// TIA Portal V19 export
VAR_GLOBAL   // PLC tag table "A03_301"
   A0301_Rulliera_Phc_1 AT %I201.2 : Bool;   // 1445BF1
   A0301_Rulliera_Phc_2 AT %I201.3 : Bool;   // 1445SQ1/SQ2/SQ3/SQ4
   A0301_Rulliera_Phc_3 AT %I201.4 : Bool;   // 1445SQ5/SQ6/SQ7/SQ8
   A0301_Rulliera_Phc_4 AT %I201.5 : Bool;   // 1446SQ1/SQ2/SQ3/SQ4
   A0301_Rulliera_Phc_5 AT %I201.6 : Bool;   // 1446BF1
   A0301_Spintore_1_Verticale_Ls_Rest AT %I201.7 : Bool;   // 1450SQ1
   A0301_Spintore_1_Verticale_V_Rest AT %Q210.0 : Bool;   // 1450YV1
   A0301_Spintore_1_Verticale_V_Work AT %Q210.1 : Bool;   // 1450YV2
   A0301_Spintore_1_Laterale_Ls_Rest AT %I202.0 : Bool;   // 1450SQ2
   A0301_Spintore_1_Laterale_V_Rest AT %Q210.2 : Bool;   // 1450YV3
   A0301_Spintore_1_Laterale_V_Work AT %Q210.3 : Bool;   // 1450YV4
   A0301_Spintore_1_Laterale_Ls_Work AT %I202.1 : Bool;   // 1450SQ3
   A0301_Spintore_2_Verticale_Ls_Rest AT %I202.2 : Bool;   // 1451SQ1
   A0301_Spintore_2_Verticale_V_Rest AT %Q210.4 : Bool;   // 1451YV1
   A0301_Spintore_2_Verticale_V_Work AT %Q210.5 : Bool;   // 1451YV2
   A0301_Spintore_2_Laterale_Ls_Rest AT %I202.3 : Bool;   // 1451SQ2
   A0301_Spintore_2_Laterale_V_Rest AT %Q210.6 : Bool;   // 1451YV3
   A0301_Spintore_2_Laterale_V_Work AT %Q210.7 : Bool;   // 1451YV4
   A0301_Spintore_2_Laterale_Ls_Work AT %I202.4 : Bool;   // 1451SQ3
   A0301_Spintore_3_Verticale_Ls_Rest AT %I202.5 : Bool;   // 1452SQ1
   A0301_Spintore_3_Verticale_V_Rest AT %Q211.0 : Bool;   // 1452YV1
   A0301_Spintore_3_Verticale_V_Work AT %Q211.1 : Bool;   // 1452YV2
   A0301_Spintore_3_Laterale_Ls_Rest AT %I202.6 : Bool;   // 1452SQ2
   A0301_Spintore_3_Laterale_V_Rest AT %Q211.2 : Bool;   // 1452YV3
   A0301_Spintore_3_Laterale_V_Work AT %Q211.3 : Bool;   // 1452YV4
   A0301_Spintore_3_Laterale_Ls_Work AT %I202.7 : Bool;   // 1452SQ3
   A0301_Spintore_4_Verticale_Ls_Rest AT %I203.0 : Bool;   // 1453SQ1
   A0301_Spintore_4_Verticale_V_Rest AT %Q211.4 : Bool;   // 1453YV1
   A0301_Spintore_4_Verticale_V_Work AT %Q211.5 : Bool;   // 1453YV2
   A0301_Spintore_4_Laterale_Ls_Rest AT %I203.1 : Bool;   // 1453SQ2
   A0301_Spintore_4_Laterale_V_Rest AT %Q211.6 : Bool;   // 1453YV3
   A0301_Spintore_4_Laterale_V_Work AT %Q211.7 : Bool;   // 1453YV4
   A0301_Spintore_4_Laterale_Ls_Work AT %I203.2 : Bool;   // 1453SQ3
   A0301_Spintore_5_Verticale_Ls_Rest AT %I203.3 : Bool;   // 1454SQ1
   A0301_Spintore_5_Verticale_V_Rest AT %Q212.0 : Bool;   // 1454YV1
   A0301_Spintore_5_Verticale_V_Work AT %Q212.1 : Bool;   // 1454YV2
   A0301_Spintore_5_Laterale_Ls_Rest AT %I203.4 : Bool;   // 1454SQ2
   A0301_Spintore_5_Laterale_V_Rest AT %Q212.2 : Bool;   // 1454YV3
   A0301_Spintore_5_Laterale_V_Work AT %Q212.3 : Bool;   // 1454YV4
   A0301_Spintore_5_Laterale_Ls_Work AT %I203.5 : Bool;   // 1454SQ3
   A0301_Spintore_6_Verticale_Ls_Rest AT %I203.6 : Bool;   // 1455SQ1
   A0301_Spintore_6_Verticale_V_Rest AT %Q212.4 : Bool;   // 1455YV1
   A0301_Spintore_6_Verticale_V_Work AT %Q212.5 : Bool;   // 1455YV2
   A0301_Spintore_6_Laterale_Ls_Rest AT %I203.7 : Bool;   // 1455SQ2
   A0301_Spintore_6_Laterale_V_Rest AT %Q212.6 : Bool;   // 1455YV3
   A0301_Spintore_6_Laterale_V_Work AT %Q212.7 : Bool;   // 1455YV4
   A0301_Spintore_6_Laterale_Ls_Work AT %I204.0 : Bool;   // 1455SQ3
   A0301_Scivolo_1_Phc_1 AT %I204.1 : Bool;   // 1470SQ1
   A0301_Scivolo_1_Phc_2 AT %I204.2 : Bool;   // 1470SQ2
   A0301_Scivolo_1_Phc_3 AT %I204.3 : Bool;   // 1470SQ3
   A0301_Scivolo_1_Phc_4 AT %I204.4 : Bool;   // 1470SQ4
   A0301_Cinghia_1_Phc_1 AT %I253.0 : Bool;   // 1510SQ1
   A0301_Cinghia_1_Phc_4 AT %I253.3 : Bool;   // 1510SQ4
   A0301_Cinghia_1_Phc_2 AT %I253.1 : Bool;   // 1510SQ2
   A0301_Cinghia_1_Phc_3 AT %I253.2 : Bool;   // 1510SQ3
   A0301_Cinghia_1_Phc_5 AT %I253.4 : Bool;   // 1510SQ5
   A0301_Cinghia_1_Phc_6 AT %I253.5 : Bool;   // 1510SQ6
   A0301_Cinghia_1_Phc_7 AT %I253.6 : Bool;   // 1510SQ7
   A0301_Cinghia_1_Phc_8 AT %I253.7 : Bool;   // 1510SQ8
   A0301_Cinghia_2_Phc_1 AT %I254.0 : Bool;   // 1511SQ1
   A0301_Cinghia_2_Phc_2 AT %I254.1 : Bool;   // 1511SQ2
   A0301_Cinghia_2_Phc_3 AT %I254.2 : Bool;   // 1511SQ3
   A0301_Cinghia_2_Phc_4 AT %I254.3 : Bool;   // 1511SQ4
   A0301_Cinghia_2_Phc_5 AT %I254.4 : Bool;   // 1511SQ5
   A0301_Cinghia_2_Phc_6 AT %I254.5 : Bool;   // 1511SQ6
   A0301_Cinghia_2_Phc_7 AT %I254.6 : Bool;   // 1511SQ7
   A0301_Cinghia_2_Phc_8 AT %I254.7 : Bool;   // 1511SQ8
   A0301_Cinghia_4_Phc_1 AT %I255.0 : Bool;   // 1513SQ1
   A0301_Cinghia_4_Phc_2 AT %I255.1 : Bool;   // 1513SQ2
   A0301_Cinghia_4_Phc_3 AT %I255.2 : Bool;   // 1513SQ3
   A0301_Cinghia_4_Phc_4 AT %I255.3 : Bool;   // 1513SQ4
   A0301_Cinghia_4_Phc_5 AT %I255.4 : Bool;   // 1513SQ5
   A0301_Cinghia_4_Phc_6 AT %I255.5 : Bool;   // 1513SQ6
   A0301_Cinghia_4_Phc_7 AT %I255.6 : Bool;   // 1513SQ7
   A0301_Cinghia_4_Phc_8 AT %I255.7 : Bool;   // 1513SQ8
   "A0301_CinghiaTrasporto_1.1_Ls_Rest_1" AT %I256.0 : Bool;   // 1530SQ1
   "A0301_CinghiaTrasporto_1.1_Ls_Work_2" AT %I256.1 : Bool;   // 1530SQ2
   "A0301_CinghiaTrasporto_1.1_Ls_Rest_3" AT %I256.2 : Bool;   // 1530SQ3
   "A0301_CinghiaTrasporto_1.1_Ls_Work_4" AT %I256.3 : Bool;   // 1530SQ4
   "A0301_CinghiaTrasporto_1.1_Ls_Rest_5" AT %I256.4 : Bool;   // 1530SQ5
   "A0301_CinghiaTrasporto_1.1_Ls_Work_6" AT %I256.5 : Bool;   // 1530SQ6
   "A0301_CinghiaTrasporto_1.1_Ls_Rest_7" AT %I256.6 : Bool;   // 1530SQ7
   "A0301_CinghiaTrasporto_1.2_Ls_Rest_1" AT %I257.0 : Bool;   // 1531SQ1
   "A0301_CinghiaTrasporto_1.2_Ls_Work_2" AT %I257.1 : Bool;   // 1531SQ2
   "A0301_CinghiaTrasporto_1.2_Ls_Rest_3" AT %I257.2 : Bool;   // 1531SQ3
   "A0301_CinghiaTrasporto_1.2_Ls_Work_4" AT %I257.3 : Bool;   // 1531SQ4
   "A0301_CinghiaTrasporto_1.2_Ls_Rest_5" AT %I257.4 : Bool;   // 1531SQ5
   "A0301_CinghiaTrasporto_2.1_Ls_Rest_1" AT %I258.0 : Bool;   // 1532SQ1
   "A0301_CinghiaTrasporto_2.1_Ls_Work_2" AT %I258.1 : Bool;   // 1532SQ2
   "A0301_CinghiaTrasporto_2.1_Ls_Rest_3" AT %I258.2 : Bool;   // 1532SQ3
   "A0301_CinghiaTrasporto_2.1_Ls_Work_4" AT %I258.3 : Bool;   // 1532SQ4
   "A0301_CinghiaTrasporto_2.1_Ls_Rest_5" AT %I258.4 : Bool;   // 1532SQ5
   "A0301_CinghiaTrasporto_2.1_Ls_Work_6" AT %I258.5 : Bool;   // 1532SQ6
   "A0301_CinghiaTrasporto_2.1_Ls_Rest_7" AT %I258.6 : Bool;   // 1532SQ7
   "A0301_CinghiaTrasporto_2.2_Ls_Rest_1" AT %I259.0 : Bool;   // 1533SQ1
   "A0301_CinghiaTrasporto_2.2_Ls_Work_2" AT %I259.1 : Bool;   // 1533SQ2
   "A0301_CinghiaTrasporto_2.2_Ls_Rest_3" AT %I259.2 : Bool;   // 1533SQ3
   "A0301_CinghiaTrasporto_2.2_Ls_Work_4" AT %I259.3 : Bool;   // 1533SQ4
   "A0301_CinghiaTrasporto_2.2_Ls_Rest_5" AT %I259.4 : Bool;   // 1533SQ5
   "A0301_CinghiaTrasporto_3.1_Ls_Rest_1" AT %I260.0 : Bool;   // 1534SQ1
   "A0301_CinghiaTrasporto_3.1_Ls_Work_2" AT %I260.1 : Bool;   // 1534SQ2
   "A0301_CinghiaTrasporto_3.1_Ls_Rest_3" AT %I260.2 : Bool;   // 1534SQ3
   "A0301_CinghiaTrasporto_3.1_Ls_Work_4" AT %I260.3 : Bool;   // 1534SQ4
   "A0301_CinghiaTrasporto_3.1_Ls_Rest_5" AT %I260.4 : Bool;   // 1534SQ5
   "A0301_CinghiaTrasporto_3.1_Ls_Work_6" AT %I260.5 : Bool;   // 1534SQ6
   "A0301_CinghiaTrasporto_3.1_Ls_Rest_7" AT %I260.6 : Bool;   // 1534SQ7
   A0301_SpintoreLaterale_2_V_Work_2 AT %Q273.3 : Bool;   // 1574YV4
   A0301_SpintoreLaterale_2_V_Work_1 AT %Q273.1 : Bool;   // 1574YV2
   A0301_SpintoreLaterale_2_V_Rest_2 AT %Q273.2 : Bool;   // 1574YV3
   A0301_SpintoreLaterale_2_V_Rest_1 AT %Q273.0 : Bool;   // 1574YV1
   A0301_SpintoreLaterale_2_Ls_Work_2 AT %I269.0 : Bool;   // 1574SQ4
   A0301_SpintoreLaterale_2_Ls_Work_1 AT %I268.6 : Bool;   // 1574SQ2
   A0301_SpintoreLaterale_2_Ls_Rest_2 AT %I268.7 : Bool;   // 1574SQ3
   A0301_SpintoreLaterale_2_Ls_Rest_1 AT %I268.5 : Bool;   // 1574SQ1
   A0301_SpintoreLaterale_1_V_Work_2 AT %Q260.7 : Bool;   // 1570YV4
   A0301_SpintoreLaterale_1_V_Work_1 AT %Q260.5 : Bool;   // 1570YV2
   A0301_SpintoreLaterale_1_V_Rest_2 AT %Q260.6 : Bool;   // 1570YV3
   A0301_SpintoreLaterale_1_V_Rest_1 AT %Q260.4 : Bool;   // 1570YV1
   A0301_SpintoreLaterale_1_Ls_Work_2 AT %I268.4 : Bool;   // 1570SQ4
   A0301_SpintoreLaterale_1_Ls_Work_1 AT %I268.2 : Bool;   // 1570SQ2
   A0301_SpintoreLaterale_1_Ls_Rest_2 AT %I268.3 : Bool;   // 1570SQ3
   A0301_SpintoreLaterale_1_Ls_Rest_1 AT %I268.1 : Bool;   // 1570SQ1
   A0301_Ribaltatore_Ls_Minimo AT %I252.7 : Bool;   // 1562SQ1
   A0301_Ribaltatore_Ls_Massimo AT %I268.0 : Bool;   // 1562SQ2
   "A0301_CinghiaTrasporto_6.2_V_Work_4" AT %Q272.3 : Bool;   // 1541YV4
   "A0301_CinghiaTrasporto_6.2_V_Work_2" AT %Q272.1 : Bool;   // 1541YV2
   "A0301_CinghiaTrasporto_6.2_V_Rest_5" AT %Q272.4 : Bool;   // 1541YV5
   "A0301_CinghiaTrasporto_6.2_V_Rest_3" AT %Q272.2 : Bool;   // 1541YV3
   "A0301_CinghiaTrasporto_6.2_V_Rest_1" AT %Q272.0 : Bool;   // 1541YV1
   "A0301_CinghiaTrasporto_6.2_Ls_Work_4" AT %I267.3 : Bool;   // 1541SQ4
   "A0301_CinghiaTrasporto_6.2_Ls_Work_2" AT %I267.1 : Bool;   // 1541SQ2
   "A0301_CinghiaTrasporto_6.2_Ls_Rest_5" AT %I267.4 : Bool;   // 1541SQ5
   "A0301_CinghiaTrasporto_6.2_Ls_Rest_3" AT %I267.2 : Bool;   // 1541SQ3
   "A0301_CinghiaTrasporto_6.2_Ls_Rest_1" AT %I267.0 : Bool;   // 1541SQ1
   "A0301_CinghiaTrasporto_6.1_V_Work_6" AT %Q271.5 : Bool;   // 1540YV6
   "A0301_CinghiaTrasporto_6.1_V_Work_4" AT %Q271.3 : Bool;   // 1540YV4
   "A0301_CinghiaTrasporto_6.1_V_Work_2" AT %Q271.1 : Bool;   // 1540YV2
   "A0301_CinghiaTrasporto_6.1_V_Rest_7" AT %Q271.6 : Bool;   // 1540YV7
   "A0301_CinghiaTrasporto_6.1_V_Rest_5" AT %Q271.4 : Bool;   // 1540YV5
   "A0301_CinghiaTrasporto_6.1_V_Rest_3" AT %Q271.2 : Bool;   // 1540YV3
   "A0301_CinghiaTrasporto_6.1_V_Rest_1" AT %Q271.0 : Bool;   // 1540YV1
   "A0301_CinghiaTrasporto_6.1_Ls_Work_6" AT %I266.5 : Bool;   // 1540SQ6
   "A0301_CinghiaTrasporto_6.1_Ls_Work_4" AT %I266.3 : Bool;   // 1540SQ4
   "A0301_CinghiaTrasporto_6.1_Ls_Work_2" AT %I266.1 : Bool;   // 1540SQ2
   "A0301_CinghiaTrasporto_6.1_Ls_Rest_7" AT %I266.6 : Bool;   // 1540SQ7
   "A0301_CinghiaTrasporto_6.1_Ls_Rest_5" AT %I266.4 : Bool;   // 1540SQ5
   "A0301_CinghiaTrasporto_6.1_Ls_Rest_3" AT %I266.2 : Bool;   // 1540SQ3
   "A0301_CinghiaTrasporto_6.1_Ls_Rest_1" AT %I266.0 : Bool;   // 1540SQ1
   "A0301_CinghiaTrasporto_5.2_V_Work_4" AT %Q270.3 : Bool;   // 1539YV4
   "A0301_CinghiaTrasporto_5.2_V_Work_2" AT %Q270.1 : Bool;   // 1539YV2
   "A0301_CinghiaTrasporto_5.2_V_Rest_5" AT %Q270.4 : Bool;   // 1539YV5
   "A0301_CinghiaTrasporto_5.2_V_Rest_3" AT %Q270.2 : Bool;   // 1539YV3
   "A0301_CinghiaTrasporto_5.2_V_Rest_1" AT %Q270.0 : Bool;   // 1539YV1
   "A0301_CinghiaTrasporto_5.2_Ls_Work_4" AT %I265.3 : Bool;   // 1539SQ4
   "A0301_CinghiaTrasporto_5.2_Ls_Work_2" AT %I265.1 : Bool;   // 1539SQ2
   "A0301_CinghiaTrasporto_5.2_Ls_Rest_5" AT %I265.4 : Bool;   // 1539SQ5
   "A0301_CinghiaTrasporto_5.2_Ls_Rest_3" AT %I265.2 : Bool;   // 1539SQ3
   "A0301_CinghiaTrasporto_5.2_Ls_Rest_1" AT %I265.0 : Bool;   // 1539SQ1
   "A0301_CinghiaTrasporto_5.1_V_Work_6" AT %Q269.5 : Bool;   // 1538YV6
   "A0301_CinghiaTrasporto_5.1_V_Work_4" AT %Q269.3 : Bool;   // 1538YV4
   "A0301_CinghiaTrasporto_5.1_V_Work_2" AT %Q269.1 : Bool;   // 1538YV2
   "A0301_CinghiaTrasporto_5.1_V_Rest_7" AT %Q269.6 : Bool;   // 1538YV7
   "A0301_CinghiaTrasporto_5.1_V_Rest_5" AT %Q269.4 : Bool;   // 1538YV5
   "A0301_CinghiaTrasporto_5.1_V_Rest_3" AT %Q269.2 : Bool;   // 1538YV3
   "A0301_CinghiaTrasporto_5.1_V_Rest_1" AT %Q269.0 : Bool;   // 1538YV1
   "A0301_CinghiaTrasporto_5.1_Ls_Work_6" AT %I264.5 : Bool;   // 1538SQ6
   "A0301_CinghiaTrasporto_5.1_Ls_Work_4" AT %I264.3 : Bool;   // 1538SQ4
   "A0301_CinghiaTrasporto_5.1_Ls_Work_2" AT %I264.1 : Bool;   // 1538SQ2
   "A0301_CinghiaTrasporto_5.1_Ls_Rest_7" AT %I264.6 : Bool;   // 1538SQ7
   "A0301_CinghiaTrasporto_5.1_Ls_Rest_5" AT %I264.4 : Bool;   // 1538SQ5
   "A0301_CinghiaTrasporto_5.1_Ls_Rest_3" AT %I264.2 : Bool;   // 1538SQ3
   "A0301_CinghiaTrasporto_5.1_Ls_Rest_1" AT %I264.0 : Bool;   // 1538SQ1
   "A0301_CinghiaTrasporto_4.2_V_Work_4" AT %Q268.3 : Bool;   // 1537YV4
   "A0301_CinghiaTrasporto_4.2_V_Work_2" AT %Q268.1 : Bool;   // 1537YV2
   "A0301_CinghiaTrasporto_4.2_V_Rest_5" AT %Q268.4 : Bool;   // 1537YV5
   "A0301_CinghiaTrasporto_4.2_V_Rest_3" AT %Q268.2 : Bool;   // 1537YV3
   "A0301_CinghiaTrasporto_4.2_V_Rest_1" AT %Q268.0 : Bool;   // 1537YV1
   "A0301_CinghiaTrasporto_4.2_Ls_Work_4" AT %I263.3 : Bool;   // 1537SQ4
   "A0301_CinghiaTrasporto_4.2_Ls_Work_2" AT %I263.1 : Bool;   // 1537SQ2
   "A0301_CinghiaTrasporto_4.2_Ls_Rest_5" AT %I263.4 : Bool;   // 1537SQ5
   "A0301_CinghiaTrasporto_4.2_Ls_Rest_3" AT %I263.2 : Bool;   // 1537SQ3
   "A0301_CinghiaTrasporto_4.2_Ls_Rest_1" AT %I263.0 : Bool;   // 1537SQ1
   "A0301_CinghiaTrasporto_4.1_V_Work_6" AT %Q267.5 : Bool;   // 1536YV6
   "A0301_CinghiaTrasporto_4.1_V_Work_4" AT %Q267.3 : Bool;   // 1536YV4
   "A0301_CinghiaTrasporto_4.1_V_Work_2" AT %Q267.1 : Bool;   // 1536YV2
   "A0301_CinghiaTrasporto_4.1_V_Rest_7" AT %Q267.6 : Bool;   // 1536YV7
   "A0301_CinghiaTrasporto_4.1_V_Rest_5" AT %Q267.4 : Bool;   // 1536YV5
   "A0301_CinghiaTrasporto_4.1_V_Rest_3" AT %Q267.2 : Bool;   // 1536YV3
   "A0301_CinghiaTrasporto_4.1_V_Rest_1" AT %Q267.0 : Bool;   // 1536YV1
   "A0301_CinghiaTrasporto_4.1_Ls_Work_6" AT %I262.5 : Bool;   // 1536SQ6
   "A0301_CinghiaTrasporto_4.1_Ls_Work_4" AT %I262.3 : Bool;   // 1536SQ4
   "A0301_CinghiaTrasporto_4.1_Ls_Work_2" AT %I262.1 : Bool;   // 1536SQ2
   "A0301_CinghiaTrasporto_4.1_Ls_Rest_7" AT %I262.6 : Bool;   // 1536SQ7
   "A0301_CinghiaTrasporto_4.1_Ls_Rest_5" AT %I262.4 : Bool;   // 1536SQ5
   "A0301_CinghiaTrasporto_4.1_Ls_Rest_3" AT %I262.2 : Bool;   // 1536SQ3
   "A0301_CinghiaTrasporto_4.1_Ls_Rest_1" AT %I262.0 : Bool;   // 1536SQ1
   "A0301_CinghiaTrasporto_3.2_V_Work_4" AT %Q266.3 : Bool;   // 1535YV4
   "A0301_CinghiaTrasporto_3.2_V_Work_2" AT %Q266.1 : Bool;   // 1535YV2
   "A0301_CinghiaTrasporto_3.2_V_Rest_5" AT %Q266.4 : Bool;   // 1535YV5
   "A0301_CinghiaTrasporto_3.2_V_Rest_3" AT %Q266.2 : Bool;   // 1535YV3
   "A0301_CinghiaTrasporto_3.2_V_Rest_1" AT %Q266.0 : Bool;   // 1535YV1
   "A0301_CinghiaTrasporto_3.2_Ls_Work_4" AT %I261.3 : Bool;   // 1535SQ4
   "A0301_CinghiaTrasporto_3.2_Ls_Work_2" AT %I261.1 : Bool;   // 1535SQ2
   "A0301_CinghiaTrasporto_3.2_Ls_Rest_5" AT %I261.4 : Bool;   // 1535SQ5
   "A0301_CinghiaTrasporto_3.2_Ls_Rest_3" AT %I261.2 : Bool;   // 1535SQ3
   "A0301_CinghiaTrasporto_3.2_Ls_Rest_1" AT %I261.0 : Bool;   // 1535SQ1
   "A0301_CinghiaTrasporto_3.1_V_Work_6" AT %Q265.5 : Bool;   // 1534YV6
   "A0301_CinghiaTrasporto_3.1_V_Work_4" AT %Q265.3 : Bool;   // 1534YV4
   "A0301_CinghiaTrasporto_3.1_V_Work_2" AT %Q265.1 : Bool;   // 1534YV2
   "A0301_CinghiaTrasporto_3.1_V_Rest_7" AT %Q265.6 : Bool;   // 1534YV7
   "A0301_CinghiaTrasporto_3.1_V_Rest_5" AT %Q265.4 : Bool;   // 1534YV5
   "A0301_CinghiaTrasporto_3.1_V_Rest_3" AT %Q265.2 : Bool;   // 1534YV3
   "A0301_CinghiaTrasporto_3.1_V_Rest_1" AT %Q265.0 : Bool;   // 1534YV1
   "A0301_CinghiaTrasporto_2.2_V_Work_4" AT %Q264.3 : Bool;   // 1533YV4
   "A0301_CinghiaTrasporto_2.2_V_Work_2" AT %Q264.1 : Bool;   // 1533YV2
   "A0301_CinghiaTrasporto_2.2_V_Rest_5" AT %Q264.4 : Bool;   // 1533YV5
   "A0301_CinghiaTrasporto_2.2_V_Rest_3" AT %Q264.2 : Bool;   // 1533YV3
   "A0301_CinghiaTrasporto_2.2_V_Rest_1" AT %Q264.0 : Bool;   // 1533YV1
   "A0301_CinghiaTrasporto_2.1_V_Work_6" AT %Q263.5 : Bool;   // 1532YV6
   "A0301_CinghiaTrasporto_2.1_V_Work_4" AT %Q263.3 : Bool;   // 1532YV4
   "A0301_CinghiaTrasporto_2.1_V_Work_2" AT %Q263.1 : Bool;   // 1532YV2
   "A0301_CinghiaTrasporto_2.1_V_Rest_7" AT %Q263.6 : Bool;   // 1532YV7
   "A0301_CinghiaTrasporto_2.1_V_Rest_5" AT %Q263.4 : Bool;   // 1532YV5
   "A0301_CinghiaTrasporto_2.1_V_Rest_3" AT %Q263.2 : Bool;   // 1532YV3
   "A0301_CinghiaTrasporto_2.1_V_Rest_1" AT %Q263.0 : Bool;   // 1532YV1
   "A0301_CinghiaTrasporto_1.2_V_Work_4" AT %Q262.3 : Bool;   // 1531YV4
   "A0301_CinghiaTrasporto_1.2_V_Work_2" AT %Q262.1 : Bool;   // 1531YV2
   "A0301_CinghiaTrasporto_1.2_V_Rest_5" AT %Q262.4 : Bool;   // 1531YV5
   "A0301_CinghiaTrasporto_1.2_V_Rest_3" AT %Q262.2 : Bool;   // 1531YV3
   "A0301_CinghiaTrasporto_1.2_V_Rest_1" AT %Q262.0 : Bool;   // 1531YV1
   "A0301_CinghiaTrasporto_1.1_V_Work_6" AT %Q261.5 : Bool;   // 1530YV6
   "A0301_CinghiaTrasporto_1.1_V_Work_4" AT %Q261.3 : Bool;   // 1530YV4
   "A0301_CinghiaTrasporto_1.1_V_Work_2" AT %Q261.1 : Bool;   // 1530YV2
   "A0301_CinghiaTrasporto_1.1_V_Rest_7" AT %Q261.6 : Bool;   // 1530YV7
   "A0301_CinghiaTrasporto_1.1_V_Rest_5" AT %Q261.4 : Bool;   // 1530YV5
   "A0301_CinghiaTrasporto_1.1_V_Rest_3" AT %Q261.2 : Bool;   // 1530YV3
   "A0301_CinghiaTrasporto_1.1_V_Rest_1" AT %Q261.0 : Bool;   // 1530YV1
   A0301_Sfalsatore_V_Work AT %Q260.3 : Bool;   // 1500YV4
   A0301_Sfalsatore_V_Rest AT %Q260.2 : Bool;   // 1500YV3
   A0301_Sfalsatore_Ls_Work AT %I252.6 : Bool;   // 1500SQ4
   A0301_Sfalsatore_Ls_Rest AT %I252.5 : Bool;   // 1500SQ3
   A0301_Pareggiatore_V_Work AT %Q260.1 : Bool;   // 1500YV2
   A0301_Pareggiatore_V_Rest AT %Q260.0 : Bool;   // 1500YV1
   A0301_Pareggiatore_Ls_Work AT %I252.4 : Bool;   // 1500SQ2
   A0301_Pareggiatore_Ls_Rest AT %I252.3 : Bool;   // 1500SQ1
   A0302_AI_SpintoreLaterale_1_Posizionamento AT %IW928 : Int;   // 513A1 - 1572A1
   A0302_AI_SpintoreLaterale_2_Posizionamento AT %IW930 : Int;   // 513A1 - 1576A1
   A0301_Scivolo_1_Phc_5_LIBERO AT %I204.5 : Bool;   // 147005
   A0301_Scivolo_1_Phc_6_LIBERO AT %I204.6 : Bool;   // 147006
   "A0301_CinghiaTrasporto_1.1_V_Work_8" AT %Q261.7 : Bool;   // 1530YV8
   "A0301_CinghiaTrasporto_1.2_V_Work_6" AT %Q262.5 : Bool;   // 1531YV6
   "A0301_CinghiaTrasporto_2.1_V_Work_8" AT %Q263.7 : Bool;   // 1532YV8
   "A0301_CinghiaTrasporto_2.2_V_Work_6" AT %Q264.5 : Bool;   // 1533YV6
   "A0301_CinghiaTrasporto_3.1_V_Work_8" AT %Q265.7 : Bool;   // 1534YV8
   "A0301_CinghiaTrasporto_3.2_V_Work_6" AT %Q266.5 : Bool;   // 1535YV6
   "A0301_CinghiaTrasporto_4.1_V_Work_8" AT %Q267.7 : Bool;   // 1536YV8
   "A0301_CinghiaTrasporto_4.2_V_Work_6" AT %Q268.5 : Bool;   // 1537YV6
   "A0301_CinghiaTrasporto_5.1_V_Work_8" AT %Q269.7 : Bool;   // 1538YV8
   "A0301_CinghiaTrasporto_5.2_V_Work_6" AT %Q270.5 : Bool;   // 1539YV6
   "A0301_CinghiaTrasporto_6.1_V_Work_8" AT %Q271.7 : Bool;   // 1540YV8
   "A0301_CinghiaTrasporto_6.2_V_Work_6" AT %Q272.5 : Bool;   // 1541YV6
   A0302_Centratori_Centraggio_2_Centrale_Ls_Basso AT %I310.1 : Bool;   // 2022SQ1
   A0302_Centratori_Centraggio_2_Centrale_Ls_Alto AT %I310.2 : Bool;   // 2022SQ2
   A0302_Centratori_Centraggio_2_Centrale_Ls_Aperto AT %I310.3 : Bool;   // 2022SQ3
   A0302_Centratori_Centraggio_2_Centrale_Ls_Chiuso AT %I310.4 : Bool;   // 2022SQ4
   A0302_Centratori_Centraggio_3_Testa_Ls_Basso AT %I310.5 : Bool;   // 2024SQ1
   A0302_Centratori_Centraggio_3_Testa_Ls_Alto AT %I310.6 : Bool;   // 2024SQ2
   A0302_Centratori_Centraggio_3_Testa_Ls_Aperto AT %I310.7 : Bool;   // 2024SQ3
   A0302_Centratori_Centraggio_3_Testa_Ls_Chiuso AT %I311.0 : Bool;   // 2024SQ4
END_VAR
